FUNCTION_BLOCK FB_Module_ToolHolder IMPLEMENTS I_Module
VAR_INPUT
	bEnable					: BOOL;
	bToolRotationBtn		: BOOL;
END_VAR
VAR_IN_OUT
	bToolRotationBtnLight	: BOOL;
END_VAR
VAR
	Components			: ARRAY [0..5] OF I_Component;
	
	fbACmotor			: FB_Component_ACmotor;
	
	fbToolHolderLock	: FB_Component_SingleValve;
	fbReedLock			: FB_Component_ReedSwitch;
	fbReedUnlock		: FB_Component_ReedSwitch;
	
	fbIndexBit1			: FB_Component_InductiveSensor;
	fbIndexBit2			: FB_Component_InductiveSensor;
	idx					: INT;
	bDir				: BOOL; // placeholder because this motor is single direction
	bToolRotating		: BOOL;
END_VAR

IF bEnable THEN
	fbACmotor(
		bDeviceActive 	:= GVL.bLenze1Relay,
		sName			:= 'AC motor holder',
		bEnable			:= TRUE,
		bE1jog1			:= GVL.bLenze2JogBit1,
		bE2jog2			:= GVL.bLenze2JogBit2,
		bE3DCbrake		:= GVL.bLenze2njectionBrake,
		eE4Direction	:= bDir);
		
	fbToolHolderLock(
		sName 	:= 'Holder Lock',
		bEnable := TRUE,
		bOutput := GVL.bUnlockToolHolder);
		
	fbReedLock(
		bRawSignal	:= GVL.bToolHolderUnlocked,
		tDebounce	:= T#5MS,
		tTimeout	:= T#0S,
		sName		:= 'holder locked reed',
		bEnable		:= TRUE);
		
	fbReedUnlock(
		bRawSignal	:= GVL.bToolHolderLocked,
		tDebounce	:= T#5MS,
		tTimeout	:= T#0S,
		sName		:= 'holder unlocked reed',
		bEnable		:= TRUE);
		
	fbIndexBit1(bRawSignal := GVL.bToolHolderIndexBit1,
		tDebounce 	:= T#5MS,
		tTimeout	:= T#0S,
		sName		:= 'holder index 1',
		bEnable		:= TRUE);
		
	fbIndexBit2(bRawSignal := GVL.bToolHolderIndexBit2,
		tDebounce 	:= T#5MS,
		tTimeout	:= T#0S,
		sName		:= 'holder index 2',
		bEnable		:= TRUE);
		
	Components[0] 	:= fbACmotor;
	Components[1] 	:= fbToolHolderLock;
	Components[2] 	:= fbReedLock;
	Components[3] 	:= fbReedUnlock;
	Components[4] 	:= fbIndexBit1;
	Components[5] 	:= fbIndexBit2;
	
	FOR idx := 0 TO 5 DO
    	Components[idx].M_Start();
	END_FOR;
	
	IF bToolRotationBtn THEN
		bToolRotating := TRUE;
	END_IF
	
	IF bToolRotating THEN
		bToolRotationBtnLight := TRUE;
		bToolRotating := NOT M_Switch();
	ELSE
		bToolRotationBtnLight := FALSE;
	END_IF
END_IF

METHOD M_Halt : BOOL
VAR_INPUT
END_VAR
END_METHOD

METHOD M_Lock : BOOL
VAR_INPUT
END_VAR

VAR
	eState: INT;
END_VAR
IF bEnable AND fbACmotor.eState <> E_State.BUSY THEN 
		fbToolHolderLock.M_Retract();
END_IF;
END_METHOD

METHOD M_Start : BOOL
VAR_INPUT
END_VAR
END_METHOD

METHOD M_Stop : BOOL
VAR_INPUT
END_VAR
END_METHOD

METHOD M_Switch : BOOL
VAR_INPUT
END_VAR

VAR
	tTrigger1 	: R_TRIG;
	tTrigger2 	: R_TRIG;
END_VAR
IF bEnable AND fbReedUnlock.bSensorActive THEN	
	tTrigger1(CLK := fbIndexBit1.bRisingEdge);					// triggers to detect rising edge of index bits
	tTrigger2(CLK := fbIndexBit2.bRisingEdge);
	
	fbACmotor.M_SetFreq(Frequency := E_LenzeJogFreq.F3);		// when no index bit has triggered, high speed
	
	IF tTrigger1.Q THEN											// when first index is triggered, switch to lowest speed
		fbACmotor.M_SetFreq(Frequency := E_LenzeJogFreq.F1);
	END_IF
	
	IF tTrigger2.Q THEN											// when last index bit has triggered, turn of motor
		fbACmotor.M_SetFreq(Frequency := E_LenzeJogFreq.F0FF);
		IF fbACmotor.eState <> E_State.BUSY THEN		// if motor is off, lock plate and signal operation done
			M_lock();
			M_Switch := TRUE;
		END_IF;
	END_IF
ELSE
	M_Unlock();													// unlock plate of locked and reset edges for detecting indexes
	fbIndexBit1.M_ResetEdge();
	fbIndexBit2.M_ResetEdge();
END_IF
END_METHOD

METHOD M_Unlock : BOOL
VAR_INPUT
END_VAR
IF bEnable AND fbACmotor.eState <> E_State.BUSY THEN 
		fbToolHolderLock.M_Extend();
END_IF;
END_METHOD

END_FUNCTION_BLOCK

(* stored: Version 1.1.0.1, ProductVersion 3.1.4024.15
   POU FB_Module_ToolHolder: Id {b8caeb05-c46f-4fb5-a22c-c7afa5dce2ec}, SpecialFunc None
   Method M_Halt: Id {f4fd5710-ad40-4a73-9d1f-e22168ac17cc}
   Method M_Lock: Id {be180632-11d0-40d6-9843-f03e84e63f14}
   Method M_Start: Id {d25814ce-c93f-4e9d-95a8-b52a3b6266b0}
   Method M_Stop: Id {7b921080-9dcf-40c5-a818-6ca94e76f031}
   Method M_Switch: Id {d42bd0d4-106d-41e3-8483-38e40bc74aa0}
   Method M_Unlock: Id {d0392bfa-8354-4867-a771-cbf55ec92350} *)
